{attribute 'qualified_only'}
VAR_GLOBAL
    bPatchDispenseCommissioned : BOOL := TRUE;
    bHeatStakeCommissioned     : BOOL := TRUE;
    bVisionCommissioned        : BOOL := TRUE;
    // Engineering-only mode for commissioning the validated core before the
    // three real process stations are released.
    // TEMPORARY: TRUE for current AutoCycle / Index / Support commissioning.
    // Return to FALSE before production release.
    bCoreCommissioningMode     : BOOL := FALSE;
END_VAR

(* stored: Version 1.1.0.1, ProductVersion 3.1.4026.18
   GVL GVL_PatchPress_Interface: Id {b45dd829-ca08-4f40-ae9c-30f015682d1c} *)
